FUNCTION_BLOCK INTERNAL FB_Observer_LREAL_ EXTENDS FB_Observer_LREAL
VAR_INPUT
END_VAR
VAR_OUTPUT
END_VAR
VAR
END_VAR

PROPERTY nUpdateCounter : UDINT
GET
nUpdateCounter := THIS^._nUpdateCounter;
END_GET
END_PROPERTY

END_FUNCTION_BLOCK

(* stored: Version 1.1.0.1, ProductVersion 3.1.4024.12
   POU FB_Observer_LREAL_: Id {ed241e61-c436-0cab-1624-c560dbb3c0eb}, SpecialFunc None
   Property nUpdateCounter: Id {5f1c2085-1f63-0fc4-0efd-b5711c3f8e08}
   Get Get: Id {94e60791-76ed-092b-0dd6-22fef34365ba} *)
